FUNCTION_BLOCK Conveyor_SIFB
  (* Standard: 61499-2 *)
  (* Version 0.1, 2016-00-08, hpea485, UOA *)
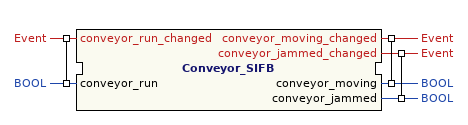
  EVENT_INPUT
    conveyor_run_changed WITH conveyor_run;
  END_EVENT
  EVENT_OUTPUT
    conveyor_moving_changed WITH conveyor_moving;
    conveyor_jammed_changed WITH conveyor_jammed;
  END_EVENT
  VAR_INPUT
    conveyor_run : BOOL;
  END_VAR
  VAR_OUTPUT
    conveyor_moving : BOOL;
    conveyor_jammed : BOOL;
  END_VAR
  VAR
    rx_conveyor_moving : BOOL; (* TOPIO_IN *)
    rx_conveyor_moving_prev : BOOL;
    rx_conveyor_jammed : BOOL; (* TOPIO_IN *)
    rx_conveyor_jammed_prev : BOOL;
    tx_conveyor_run : BOOL; (* TOPIO_OUT *)
  END_VAR
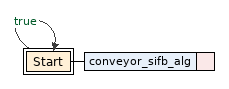
  EC_STATES
    Start : conveyor_sifb_alg;
  END_STATES
  EC_TRANSITIONS
    Start TO Start := true;
  END_TRANSITIONS
  ALGORITHM conveyor_sifb_alg IN C:
--update previous values
rx_conveyor_moving_prev <= rx_conveyor_moving;
rx_conveyor_jammed_prev <= rx_conveyor_jammed;

--these are what we use to drive events
--conveyor_moving_changed_eO_alg_out;
--conveyor_jammed_changed_eO_alg_out;

if rx_conveyor_moving_prev /= rx_conveyor_moving then
	conveyor_moving_changed_eO_alg_out <= '1';
	conveyor_moving <= rx_conveyor_moving;
end if;

if rx_conveyor_jammed_prev /= rx_conveyor_jammed then
	conveyor_jammed_changed_eO_alg_out <= '1';
	conveyor_jammed <= rx_conveyor_jammed;
end if;

--emit outputs (input is already registered to only update on tick boundary with correct input event)
tx_conveyor_run <= conveyor_run;

DONE <= '1';
  END_ALGORITHM
END_FUNCTION_BLOCK
